TYPE AlarmLimitsC :
STRUCT
END_STRUCT
END_TYPE

(* stored: Version 1.1.0.1, ProductVersion 3.1.4024.6
   DUT AlarmLimitsC: Id {3bc8872f-e1c5-4256-9155-a31ee75c44c7} *)
